PROGRAM EM02_PlacingArea_1
VAR
//----Motor-----
	// Box Placing Roller Conveyor 1	
	FB_BoxPlacingRollerConv_1			: MotorManagement;
	stBoxPlacingRollerConv_1			: stMotor;
	BoxPlacingRollerConv_1_ErrorID		: UINT;
	BoxPlacingRollerConv_1_Error		: BOOL;
	bFL_BoxPlacingRollerConv_1_Forward	: BOOL;
	bFL_BoxPlacingRollerConv_1_Reverse	: BOOL;
END_VAR

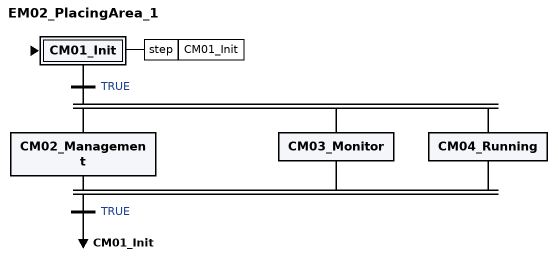
INITIAL_STEP CM01_Init:
    CM01_Init(N);  // step action
END_STEP
TRANSITION FROM CM01_Init TO (CM02_Management, CM03_Monitor, CM04_Running)
    := TRUE;
END_TRANSITION
STEP CM02_Management:
END_STEP
STEP CM03_Monitor:
END_STEP
STEP CM04_Running:
END_STEP
TRANSITION FROM (CM02_Management, CM03_Monitor, CM04_Running) TO CM01_Init
    := TRUE;
END_TRANSITION

ACTION CM01_Init:

END_ACTION

ACTION CM02_Management:
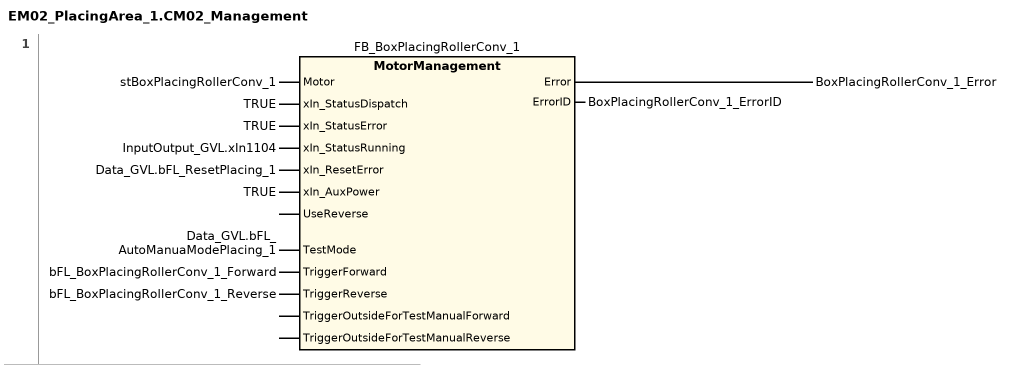
// NETWORK 1
FB_BoxPlacingRollerConv_1(
    Motor := stBoxPlacingRollerConv_1,
    xIn_StatusDispatch := TRUE,
    xIn_StatusError := TRUE,
    xIn_StatusRunning := InputOutput_GVL.xIn1104,
    xIn_ResetError := Data_GVL.bFL_ResetPlacing_1,
    xIn_AuxPower := TRUE,
    TestMode := Data_GVL.bFL_AutoManuaModePlacing_1,
    TriggerForward := bFL_BoxPlacingRollerConv_1_Forward,
    TriggerReverse := bFL_BoxPlacingRollerConv_1_Reverse,
    ErrorID => BoxPlacingRollerConv_1_ErrorID); // MotorManagement
BoxPlacingRollerConv_1_Error := FB_BoxPlacingRollerConv_1.Error;
END_ACTION

ACTION CM03_Monitor:
// NETWORK 1
END_ACTION

ACTION CM04_Running:
// NETWORK 1
END_ACTION

END_PROGRAM

(* stored: Version 1.1.0.1, ProductVersion 3.1.4024.9
   POU EM02_PlacingArea_1: Id {249a69a9-252b-4bd3-961e-1a013db347a5}, SpecialFunc None
   Action CM01_Init: Id {ef48e8a1-3ecb-4717-91ff-4b5f60424e5a}
   Action CM02_Management: Id {50f74291-9b92-4f8f-845e-b6992738adc1}
   Action CM03_Monitor: Id {8a82f764-0d44-46f5-b23a-fa321decd565}
   Action CM04_Running: Id {64115f6e-bf46-4718-9b31-6c45af0be696} *)
